Universal Robots PolyScope program: RTDE_control_2.urp

Program RTDE_control_2 (installation=default directory=/programs/new folder createdIn=5.13.1 lastSavedIn=5.13.1 robotSerialNumber=20195600129)
Calibrated DH parameters: a=[0.000295, -0.082797, -0.203177, -0.000045, 0.000063, 0]; d=[0.180731, 509.153829, -164.875613, -344.104091, 0.11995, 0.115492]; alpha=[1.57075, -0.000925, -0.000863, 1.570946, -1.569435, 0]; deltaTheta=[0, -1.396851, 0.425888, 0.970962, 0, 0]
InitVariablesNode
BeforeStart
  read_input := False
  depth_comp := False
  URCap Drive (esaDrive, ECOSPHERE Automation GmbH) dataModel(SelectedPlcDeviceNumber=0, SelectedDriveNumber=0, SelectedVelocity=0.1, SelectedAcceleration=0.4, SelectedDeceleration=0.4, SelectedMoveMode=HOMING, SelectedHomingCondition=1)
  URCap Drive (esaDrive, ECOSPHERE Automation GmbH) dataModel(SelectedPlcDeviceNumber=0, SelectedDriveNumber=1, SelectedVelocity=0.1, SelectedAcceleration=0.4, SelectedDeceleration=0.4, SelectedMoveMode=HOMING, SelectedHomingCondition=1)
  URCap Drive (esaDrive, ECOSPHERE Automation GmbH) dataModel(SelectedPlcDeviceNumber=0, SelectedDriveNumber=1, SelectedVelocity=0.1, SelectedAcceleration=0.4, SelectedDeceleration=0.4, SelectedMoveMode=MOVE_ABSOLUTE, SelectedPositionName=y_home, SelectedPosition=-0.03899)
  URCap Drive (esaDrive, ECOSPHERE Automation GmbH) dataModel(SelectedVelocity=0.1, SelectedAcceleration=0.4, SelectedDeceleration=0.4, SelectedMoveMode=MOVE_ABSOLUTE, SelectedPlcDeviceNumber=0, SelectedDriveNumber=0, SelectedPositionName=z_home, SelectedPosition=0.059)
Robot Program (runOnlyOnce=false)
  If read_input
    Set ExpressionOutput pin=digital_out[7]; expression=cut
    MoveJ speed 60 deg/s, acceleration 80 deg/s^2 (useActiveTCP=true) feature=Base
      Waypoint Variable (Variable): variable(name=tmp)
    Script: rg_grip(rg_width, rg_force,0, False ,depth_comp)
    URCap Drive (esaDrive, ECOSPHERE Automation GmbH) dataModel(SelectedPlcDeviceNumber=0, SelectedDriveNumber=1, SelectedVelocity=0.1, SelectedAcceleration=0.4, SelectedDeceleration=0.4, SelectedMoveMode=MOVE_ABSOLUTE_Variable, Variable(key=SelectedPositionVar, variable(name=y_dist)))
    If to_cut
      Set ExpressionOutput pin=digital_out[7]; expression=cut
    Script: sync()
    Script: sync()
  Script: sync()
Thread Thread_1 (runOnlyOnce=false)
  tmp := p[0,0,0,0,0,0]
  cut := False
  rg_width := 145
  rg_force := 0
  y_dist := -0.035
  to_cut := False
  Loop Forever
    Script: tmp[0] = read_input_float_register(0)
    Script: tmp[1] = read_input_float_register(1)
    Script: tmp[2] = read_input_float_register(2)
    Script: tmp[3] = read_input_float_register(3)
    Script: tmp[4] = read_input_float_register(4)
    Script: tmp[5] = read_input_float_register(5)
    Script: cut = read_input_boolean_register(73)
    Script: rg_width = read_input_float_register(8)
    Script: rg_force = read_input_float_register(9)
    Script: to_grip = read_output_boolean_register(76)
    Script: y_dist= read_input_float_register(6)
    read_input := True
    Script: sync()
